TEXTLIST TextList_Actuator_Type
  0 = '' | FR: 'Vérin de clampage' | EN: 'Clamping jack'
   = ''
END_TEXTLIST

(* stored: Version 1.1.0.1, ProductVersion 3.1.4024.10
   TextList TextList_Actuator_Type: Id {42fc7349-ffa1-4eb2-a139-3dd35dc1e381} *)
